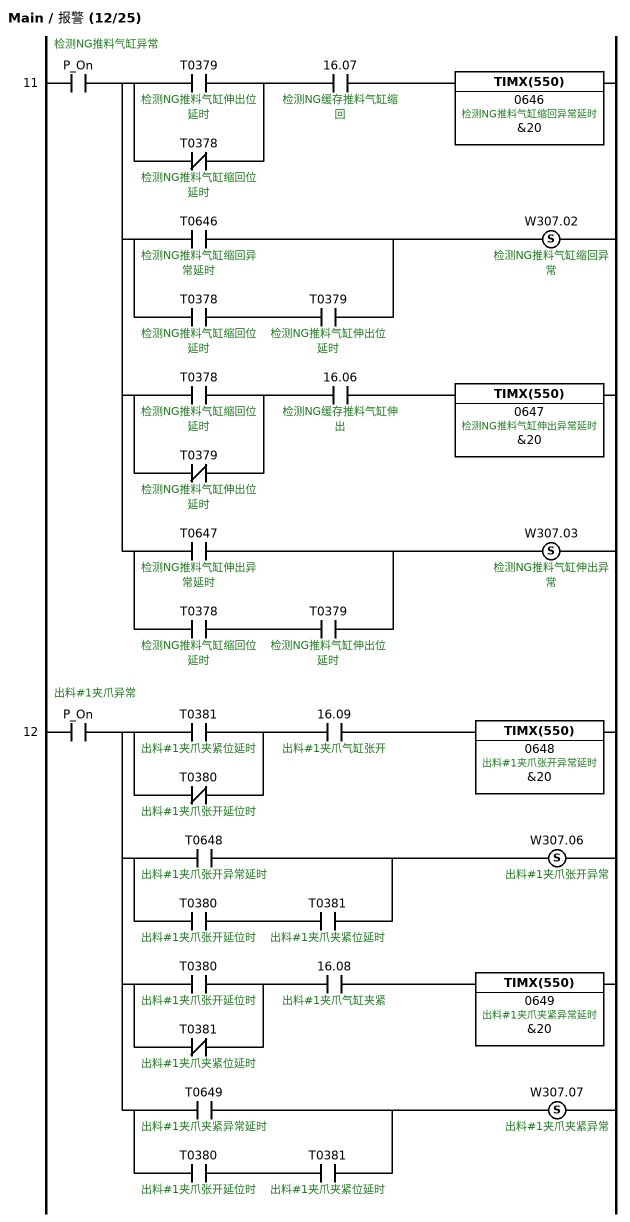
; [picture p48: Main / 报警, rungs 11-12]
; rung 11: 检测NG推料气缸异常
LD P_On
OUT TR0
LD T0379  ; 检测NG推料气缸伸出位延时
ORNOT T0378  ; 检测NG推料气缸缩回位延时
ANDLD
AND 16.07  ; 检测NG缓存推料气缸缩回
TIMX(550) 0646 &20  ; 检测NG推料气缸缩回异常延时
LD TR0
LD T0646  ; 检测NG推料气缸缩回异常延时
LD T0378  ; 检测NG推料气缸缩回位延时
AND T0379  ; 检测NG推料气缸伸出位延时
ORLD
ANDLD
SET W307.02  ; 检测NG推料气缸缩回异常
LD TR0
LD T0378  ; 检测NG推料气缸缩回位延时
ORNOT T0379  ; 检测NG推料气缸伸出位延时
ANDLD
AND 16.06  ; 检测NG缓存推料气缸伸出
TIMX(550) 0647 &20  ; 检测NG推料气缸伸出异常延时
LD TR0
LD T0647  ; 检测NG推料气缸伸出异常延时
LD T0378  ; 检测NG推料气缸缩回位延时
AND T0379  ; 检测NG推料气缸伸出位延时
ORLD
ANDLD
SET W307.03  ; 检测NG推料气缸伸出异常
; rung 12: 出料#1夹爪异常
LD P_On
OUT TR0
LD T0381  ; 出料#1夹爪夹紧位延时
ORNOT T0380  ; 出料#1夹爪张开延位时
ANDLD
AND 16.09  ; 出料#1夹爪气缸张开
TIMX(550) 0648 &20  ; 出料#1夹爪张开异常延时
LD TR0
LD T0648  ; 出料#1夹爪张开异常延时
LD T0380  ; 出料#1夹爪张开延位时
AND T0381  ; 出料#1夹爪夹紧位延时
ORLD
ANDLD
SET W307.06  ; 出料#1夹爪张开异常
LD TR0
LD T0380  ; 出料#1夹爪张开延位时
ORNOT T0381  ; 出料#1夹爪夹紧位延时
ANDLD
AND 16.08  ; 出料#1夹爪气缸夹紧
TIMX(550) 0649 &20  ; 出料#1夹爪夹紧异常延时
LD TR0
LD T0649  ; 出料#1夹爪夹紧异常延时
LD T0380  ; 出料#1夹爪张开延位时
AND T0381  ; 出料#1夹爪夹紧位延时
ORLD
ANDLD
SET W307.07  ; 出料#1夹爪夹紧异常

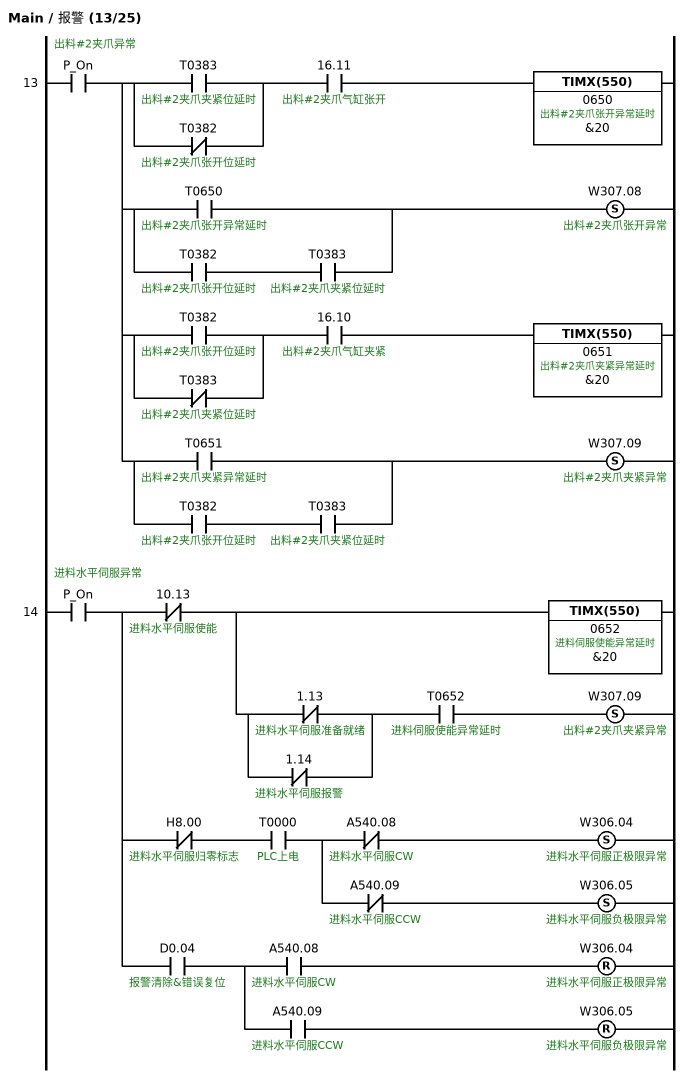
; rung 13: 出料#2夹爪异常
LD P_On
OUT TR0
LD T0383  ; 出料#2夹爪夹紧位延时
ORNOT T0382  ; 出料#2夹爪张开位延时
ANDLD
AND 16.11  ; 出料#2夹爪气缸张开
TIMX(550) 0650 &20  ; 出料#2夹爪张开异常延时
LD TR0
LD T0650  ; 出料#2夹爪张开异常延时
LD T0382  ; 出料#2夹爪张开位延时
AND T0383  ; 出料#2夹爪夹紧位延时
ORLD
ANDLD
SET W307.08  ; 出料#2夹爪张开异常
LD TR0
LD T0382  ; 出料#2夹爪张开位延时
ORNOT T0383  ; 出料#2夹爪夹紧位延时
ANDLD
AND 16.10  ; 出料#2夹爪气缸夹紧
TIMX(550) 0651 &20  ; 出料#2夹爪夹紧异常延时
LD TR0
LD T0651  ; 出料#2夹爪夹紧异常延时
LD T0382  ; 出料#2夹爪张开位延时
AND T0383  ; 出料#2夹爪夹紧位延时
ORLD
ANDLD
SET W307.09  ; 出料#2夹爪夹紧异常
; rung 14: 进料水平伺服异常
LD P_On
OUT TR0
ANDNOT 10.13  ; 进料水平伺服使能
TIMX(550) 0652 &20  ; 进料伺服使能异常延时
LDNOT 1.13  ; 进料水平伺服准备就绪
ORNOT 1.14  ; 进料水平伺服报警
ANDLD
AND T0652  ; 进料伺服使能异常延时
SET W307.09  ; 出料#2夹爪夹紧异常
LD TR0
ANDNOT H8.00  ; 进料水平伺服归零标志
AND T0000  ; PLC上电
OUT TR1
ANDNOT A540.08  ; 进料水平伺服CW
SET W306.04  ; 进料水平伺服正极限异常
LD TR1
ANDNOT A540.09  ; 进料水平伺服CCW
SET W306.05  ; 进料水平伺服负极限异常
LD TR0
AND D0.04  ; 报警清除&错误复位
OUT TR0
AND A540.08  ; 进料水平伺服CW
RSET W306.04  ; 进料水平伺服正极限异常
LD TR0
AND A540.09  ; 进料水平伺服CCW
RSET W306.05  ; 进料水平伺服负极限异常

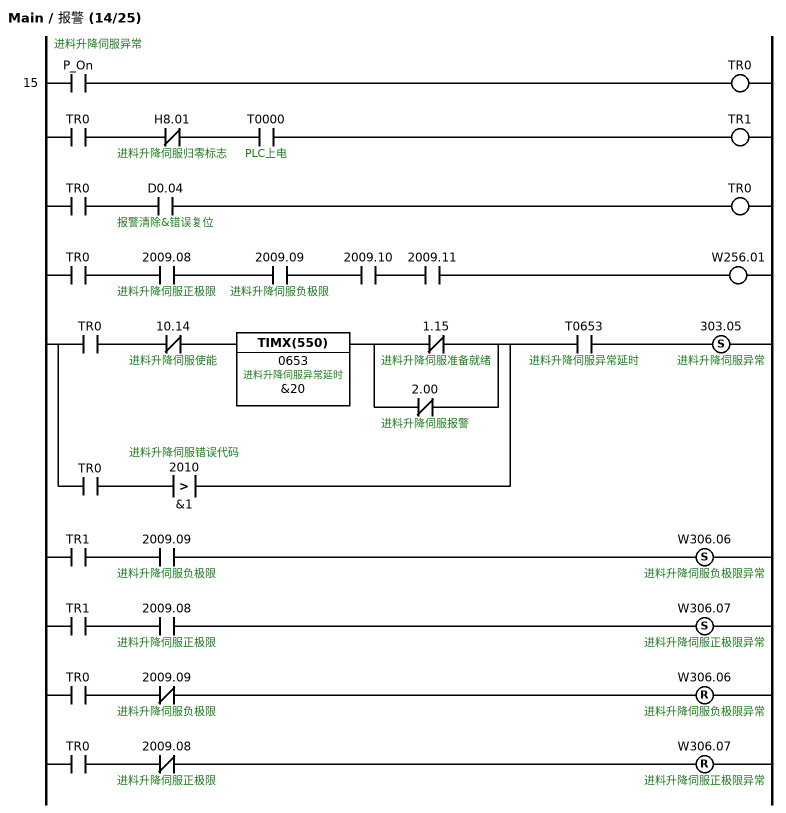
; rung 15: 进料升降伺服异常
LD P_On
OUT TR0
AND 2009.08  ; 进料升降伺服正极限
AND 2009.09  ; 进料升降伺服负极限
AND 2009.10
AND 2009.11
OUT W256.01
LD TR0
ANDNOT 10.14  ; 进料升降伺服使能
TIMX(550) 0653 &20  ; 进料升降伺服异常延时
LDNOT 1.15  ; 进料升降伺服准备就绪
ORNOT 2.00  ; 进料升降伺服报警
ANDLD
LD TR0
AND>(320) 2010 &1  ; 进料升降伺服错误代码
ORLD
AND T0653  ; 进料升降伺服异常延时
SET 303.05  ; 进料升降伺服异常
LD TR0
ANDNOT H8.01  ; 进料升降伺服归零标志
AND T0000  ; PLC上电
OUT TR1
AND 2009.09  ; 进料升降伺服负极限
SET W306.06  ; 进料升降伺服负极限异常
LD TR1
AND 2009.08  ; 进料升降伺服正极限
SET W306.07  ; 进料升降伺服正极限异常
LD TR0
AND D0.04  ; 报警清除&错误复位
OUT TR0
ANDNOT 2009.09  ; 进料升降伺服负极限
RSET W306.06  ; 进料升降伺服负极限异常
LD TR0
ANDNOT 2009.08  ; 进料升降伺服正极限
RSET W306.07  ; 进料升降伺服正极限异常

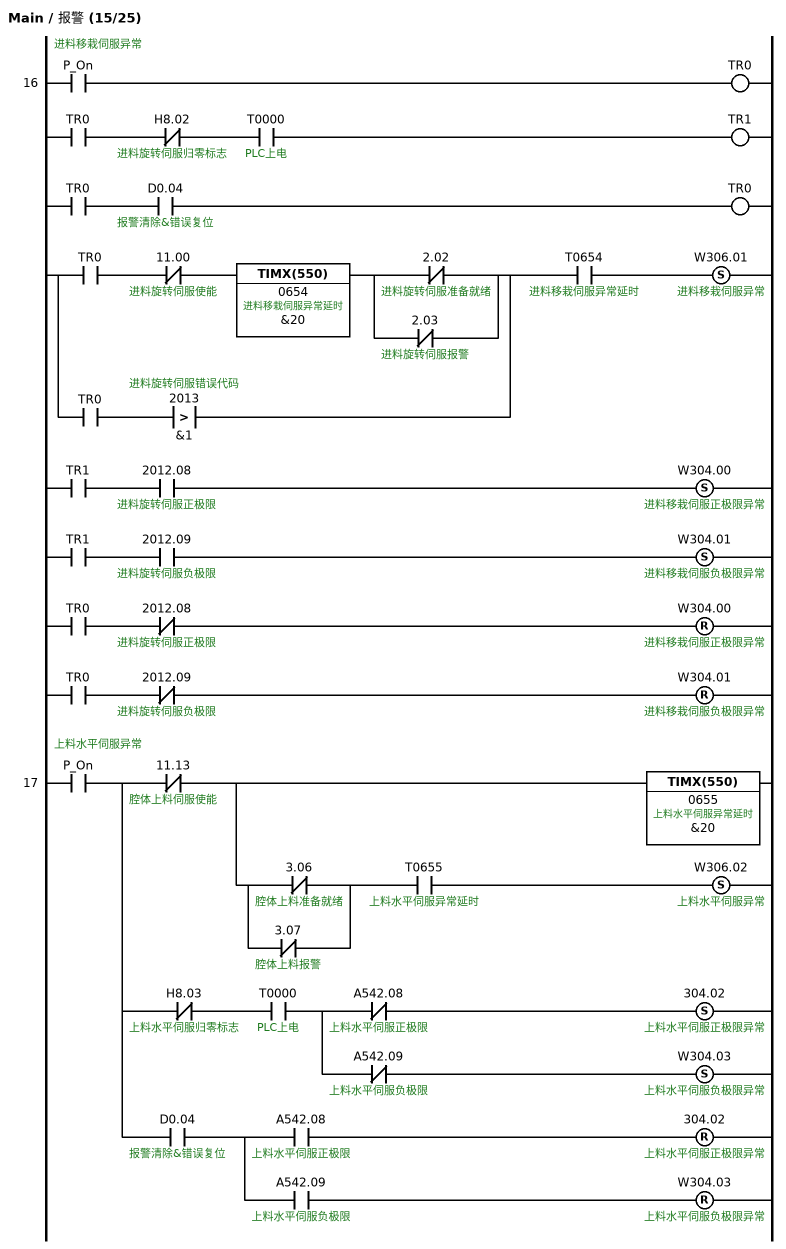
; rung 16: 进料移栽伺服异常
LD P_On
OUT TR0
ANDNOT 11.00  ; 进料旋转伺服使能
TIMX(550) 0654 &20  ; 进料移栽伺服异常延时
LDNOT 2.02  ; 进料旋转伺服准备就绪
ORNOT 2.03  ; 进料旋转伺服报警
ANDLD
LD TR0
AND>(320) 2013 &1  ; 进料旋转伺服错误代码
ORLD
AND T0654  ; 进料移栽伺服异常延时
SET W306.01  ; 进料移栽伺服异常
LD TR0
ANDNOT H8.02  ; 进料旋转伺服归零标志
AND T0000  ; PLC上电
OUT TR1
AND 2012.08  ; 进料旋转伺服正极限
SET W304.00  ; 进料移栽伺服正极限异常
LD TR1
AND 2012.09  ; 进料旋转伺服负极限
SET W304.01  ; 进料移栽伺服负极限异常
LD TR0
AND D0.04  ; 报警清除&错误复位
OUT TR0
ANDNOT 2012.08  ; 进料旋转伺服正极限
RSET W304.00  ; 进料移栽伺服正极限异常
LD TR0
ANDNOT 2012.09  ; 进料旋转伺服负极限
RSET W304.01  ; 进料移栽伺服负极限异常
; rung 17: 上料水平伺服异常
LD P_On
OUT TR0
ANDNOT 11.13  ; 腔体上料伺服使能
TIMX(550) 0655 &20  ; 上料水平伺服异常延时
LDNOT 3.06  ; 腔体上料准备就绪
ORNOT 3.07  ; 腔体上料报警
ANDLD
AND T0655  ; 上料水平伺服异常延时
SET W306.02  ; 上料水平伺服异常
LD TR0
ANDNOT H8.03  ; 上料水平伺服归零标志
AND T0000  ; PLC上电
OUT TR1
ANDNOT A542.08  ; 上料水平伺服正极限
SET 304.02  ; 上料水平伺服正极限异常
LD TR1
ANDNOT A542.09  ; 上料水平伺服负极限
SET W304.03  ; 上料水平伺服负极限异常
LD TR0
AND D0.04  ; 报警清除&错误复位
OUT TR0
AND A542.08  ; 上料水平伺服正极限
RSET 304.02  ; 上料水平伺服正极限异常
LD TR0
AND A542.09  ; 上料水平伺服负极限
RSET W304.03  ; 上料水平伺服负极限异常

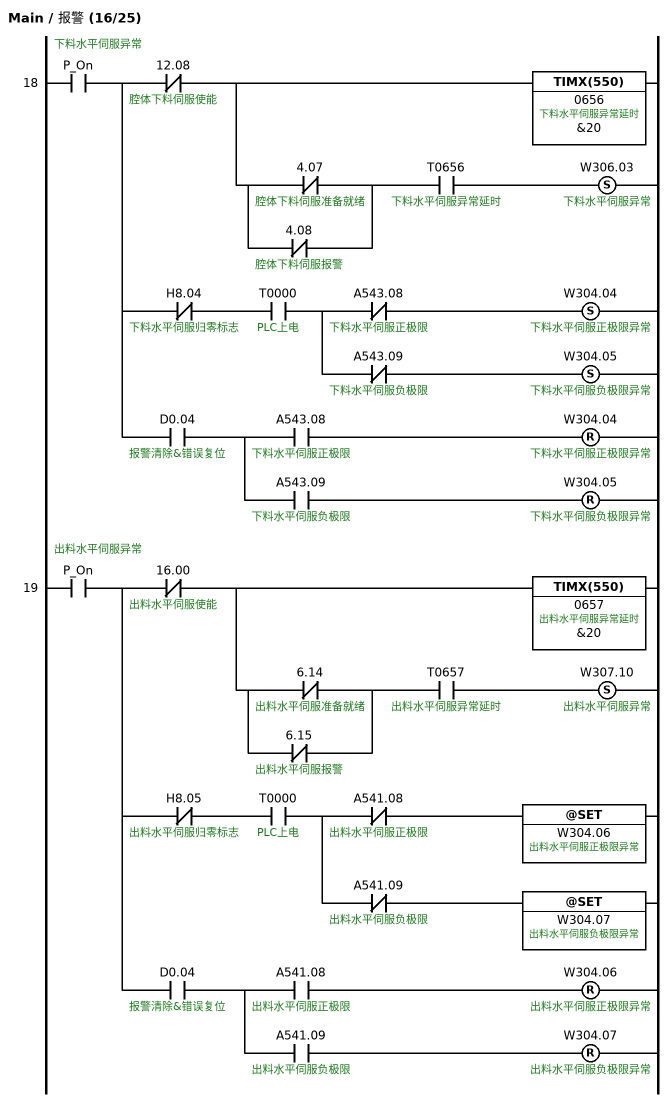
; rung 18: 下料水平伺服异常
LD P_On
OUT TR0
ANDNOT 12.08  ; 腔体下料伺服使能
TIMX(550) 0656 &20  ; 下料水平伺服异常延时
LDNOT 4.07  ; 腔体下料伺服准备就绪
ORNOT 4.08  ; 腔体下料伺服报警
ANDLD
AND T0656  ; 下料水平伺服异常延时
SET W306.03  ; 下料水平伺服异常
LD TR0
ANDNOT H8.04  ; 下料水平伺服归零标志
AND T0000  ; PLC上电
OUT TR1
ANDNOT A543.08  ; 下料水平伺服正极限
SET W304.04  ; 下料水平伺服正极限异常
LD TR1
ANDNOT A543.09  ; 下料水平伺服负极限
SET W304.05  ; 下料水平伺服负极限异常
LD TR0
AND D0.04  ; 报警清除&错误复位
OUT TR0
AND A543.08  ; 下料水平伺服正极限
RSET W304.04  ; 下料水平伺服正极限异常
LD TR0
AND A543.09  ; 下料水平伺服负极限
RSET W304.05  ; 下料水平伺服负极限异常
; rung 19: 出料水平伺服异常
LD P_On
OUT TR0
ANDNOT 16.00  ; 出料水平伺服使能
TIMX(550) 0657 &20  ; 出料水平伺服异常延时
LDNOT 6.14  ; 出料水平伺服准备就绪
ORNOT 6.15  ; 出料水平伺服报警
ANDLD
AND T0657  ; 出料水平伺服异常延时
SET W307.10  ; 出料水平伺服异常
LD TR0
ANDNOT H8.05  ; 出料水平伺服归零标志
AND T0000  ; PLC上电
OUT TR1
ANDNOT A541.08  ; 出料水平伺服正极限
@SET W304.06  ; 出料水平伺服正极限异常
LD TR1
ANDNOT A541.09  ; 出料水平伺服负极限
@SET W304.07  ; 出料水平伺服负极限异常
LD TR0
AND D0.04  ; 报警清除&错误复位
OUT TR0
AND A541.08  ; 出料水平伺服正极限
RSET W304.06  ; 出料水平伺服正极限异常
LD TR0
AND A541.09  ; 出料水平伺服负极限
RSET W304.07  ; 出料水平伺服负极限异常

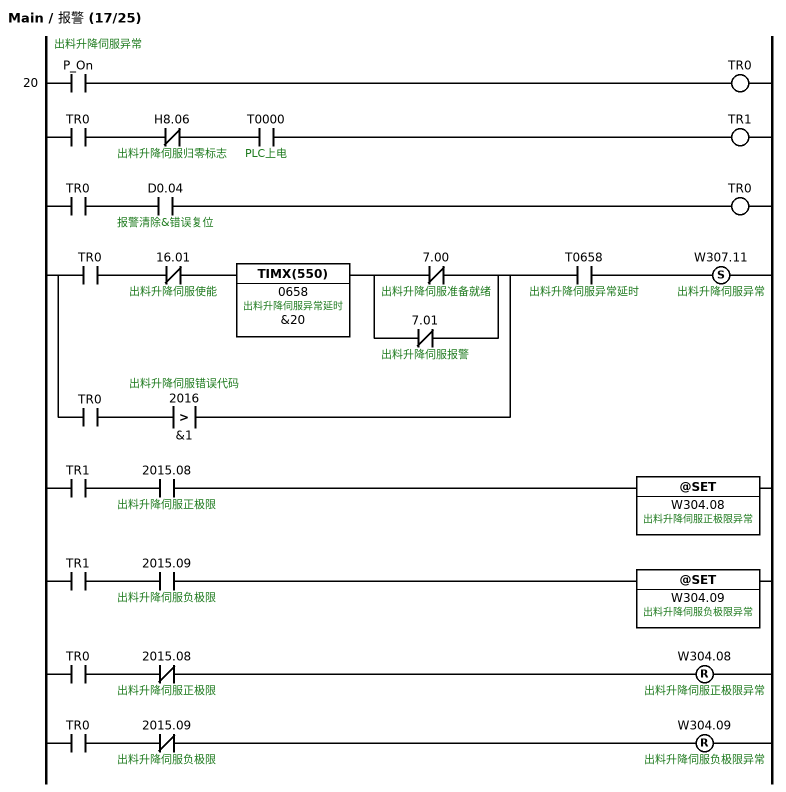
; rung 20: 出料升降伺服异常
LD P_On
OUT TR0
ANDNOT 16.01  ; 出料升降伺服使能
TIMX(550) 0658 &20  ; 出料升降伺服异常延时
LDNOT 7.00  ; 出料升降伺服准备就绪
ORNOT 7.01  ; 出料升降伺服报警
ANDLD
LD TR0
AND>(320) 2016 &1  ; 出料升降伺服错误代码
ORLD
AND T0658  ; 出料升降伺服异常延时
SET W307.11  ; 出料升降伺服异常
LD TR0
ANDNOT H8.06  ; 出料升降伺服归零标志
AND T0000  ; PLC上电
OUT TR1
AND 2015.08  ; 出料升降伺服正极限
@SET W304.08  ; 出料升降伺服正极限异常
LD TR1
AND 2015.09  ; 出料升降伺服负极限
@SET W304.09  ; 出料升降伺服负极限异常
LD TR0
AND D0.04  ; 报警清除&错误复位
OUT TR0
ANDNOT 2015.08  ; 出料升降伺服正极限
RSET W304.08  ; 出料升降伺服正极限异常
LD TR0
ANDNOT 2015.09  ; 出料升降伺服负极限
RSET W304.09  ; 出料升降伺服负极限异常

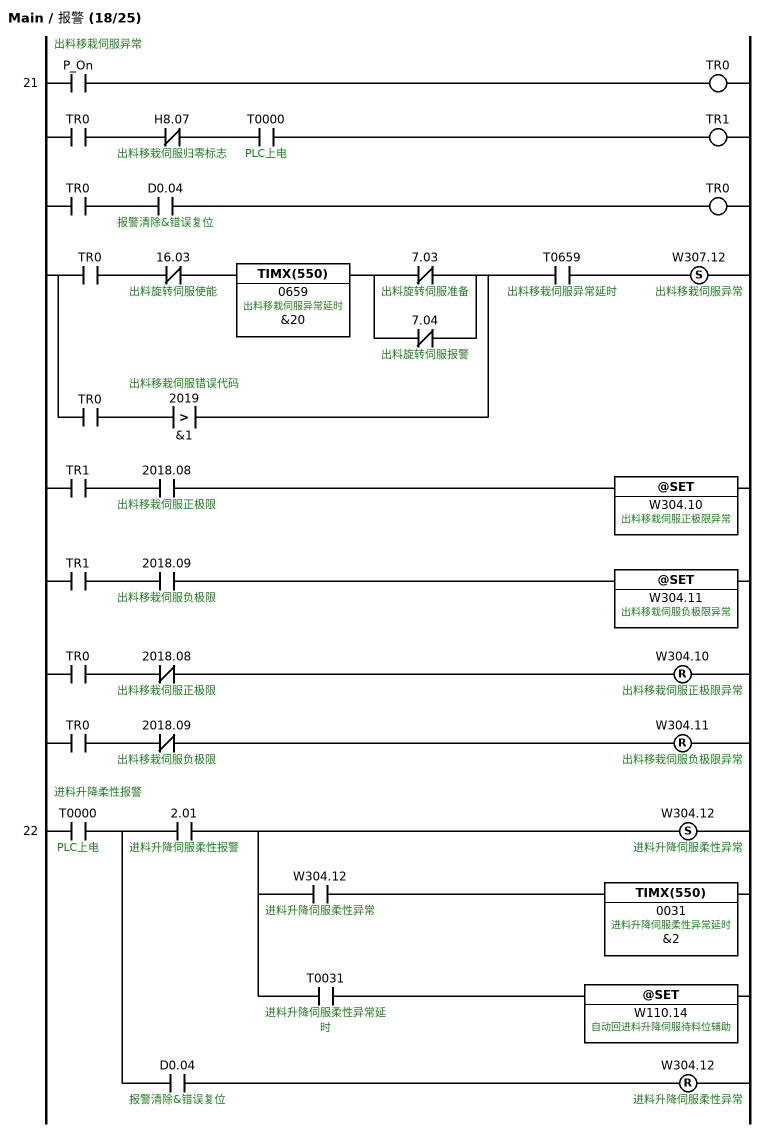
; rung 21: 出料移栽伺服异常
LD P_On
OUT TR0
ANDNOT 16.03  ; 出料旋转伺服使能
TIMX(550) 0659 &20  ; 出料移栽伺服异常延时
LDNOT 7.03  ; 出料旋转伺服准备
ORNOT 7.04  ; 出料旋转伺服报警
ANDLD
LD TR0
AND>(320) 2019 &1  ; 出料移栽伺服错误代码
ORLD
AND T0659  ; 出料移栽伺服异常延时
SET W307.12  ; 出料移栽伺服异常
LD TR0
ANDNOT H8.07  ; 出料移栽伺服归零标志
AND T0000  ; PLC上电
OUT TR1
AND 2018.08  ; 出料移栽伺服正极限
@SET W304.10  ; 出料移栽伺服正极限异常
LD TR1
AND 2018.09  ; 出料移栽伺服负极限
@SET W304.11  ; 出料移栽伺服负极限异常
LD TR0
AND D0.04  ; 报警清除&错误复位
OUT TR0
ANDNOT 2018.08  ; 出料移栽伺服正极限
RSET W304.10  ; 出料移栽伺服正极限异常
LD TR0
ANDNOT 2018.09  ; 出料移栽伺服负极限
RSET W304.11  ; 出料移栽伺服负极限异常
; rung 22: 进料升降柔性报警
LD T0000  ; PLC上电
OUT TR0
AND 2.01  ; 进料升降伺服柔性报警
OUT TR1
SET W304.12  ; 进料升降伺服柔性异常
AND W304.12  ; 进料升降伺服柔性异常
TIMX(550) 0031 &2  ; 进料升降伺服柔性异常延时
LD TR1
AND T0031  ; 进料升降伺服柔性异常延时
@SET W110.14  ; 自动回进料升降伺服待料位辅助
LD TR0
AND D0.04  ; 报警清除&错误复位
RSET W304.12  ; 进料升降伺服柔性异常

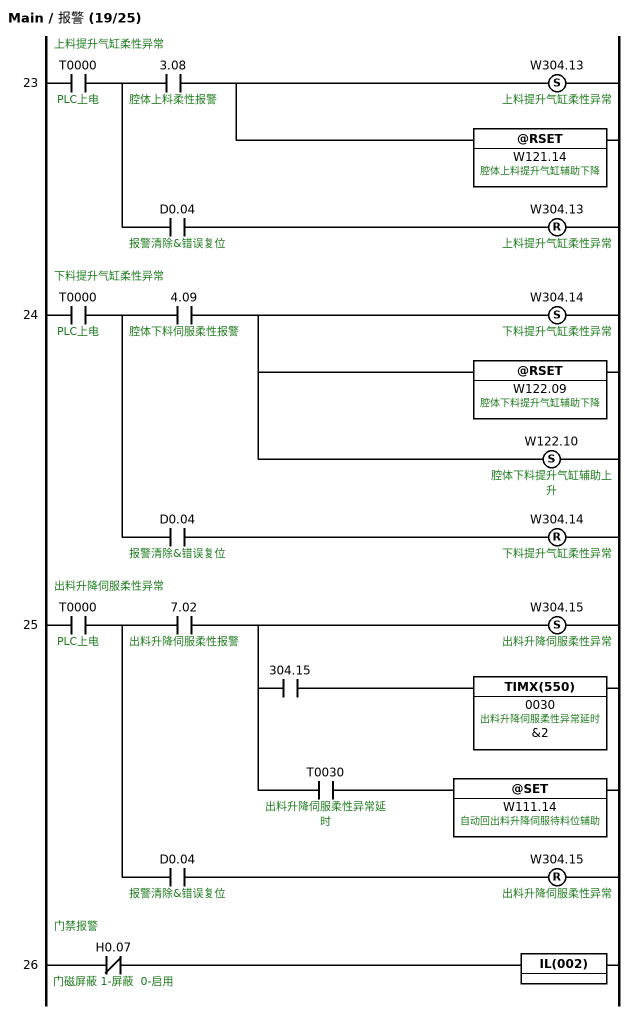
; rung 23: 上料提升气缸柔性异常
LD T0000  ; PLC上电
OUT TR0
AND 3.08  ; 腔体上料柔性报警
SET W304.13  ; 上料提升气缸柔性异常
@RSET W121.14  ; 腔体上料提升气缸辅助下降
LD TR0
AND D0.04  ; 报警清除&错误复位
RSET W304.13  ; 上料提升气缸柔性异常
; rung 24: 下料提升气缸柔性异常
LD T0000  ; PLC上电
OUT TR0
AND 4.09  ; 腔体下料伺服柔性报警
SET W304.14  ; 下料提升气缸柔性异常
@RSET W122.09  ; 腔体下料提升气缸辅助下降
SET W122.10  ; 腔体下料提升气缸辅助上升
LD TR0
AND D0.04  ; 报警清除&错误复位
RSET W304.14  ; 下料提升气缸柔性异常
; rung 25: 出料升降伺服柔性异常
LD T0000  ; PLC上电
OUT TR0
AND 7.02  ; 出料升降伺服柔性报警
OUT TR1
SET W304.15  ; 出料升降伺服柔性异常
AND 304.15
TIMX(550) 0030 &2  ; 出料升降伺服柔性异常延时
LD TR1
AND T0030  ; 出料升降伺服柔性异常延时
@SET W111.14  ; 自动回出料升降伺服待料位辅助
LD TR0
AND D0.04  ; 报警清除&错误复位
RSET W304.15  ; 出料升降伺服柔性异常
; rung 26: 门禁报警
LDNOT H0.07  ; 门磁屏蔽 1-屏蔽  0-启用
IL(002)

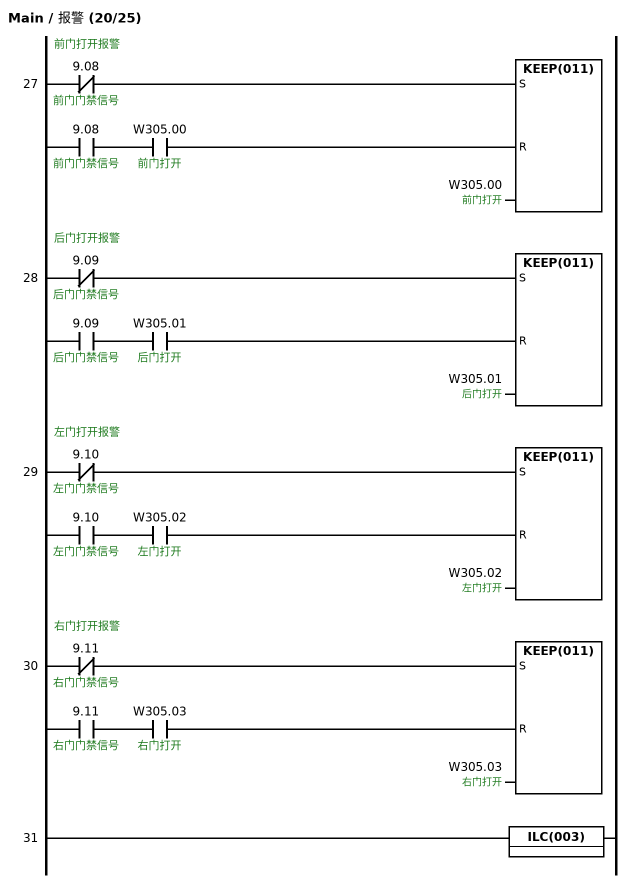
; rung 27: 前门打开报警
LDNOT 9.08  ; 前门门禁信号
LD 9.08  ; 前门门禁信号
AND W305.00  ; 前门打开
KEEP(011) W305.00  ; 前门打开
; rung 28: 后门打开报警
LDNOT 9.09  ; 后门门禁信号
LD 9.09  ; 后门门禁信号
AND W305.01  ; 后门打开
KEEP(011) W305.01  ; 后门打开
; rung 29: 左门打开报警
LDNOT 9.10  ; 左门门禁信号
LD 9.10  ; 左门门禁信号
AND W305.02  ; 左门打开
KEEP(011) W305.02  ; 左门打开
; rung 30: 右门打开报警
LDNOT 9.11  ; 右门门禁信号
LD 9.11  ; 右门门禁信号
AND W305.03  ; 右门打开
KEEP(011) W305.03  ; 右门打开
; rung 31
ILC(003)

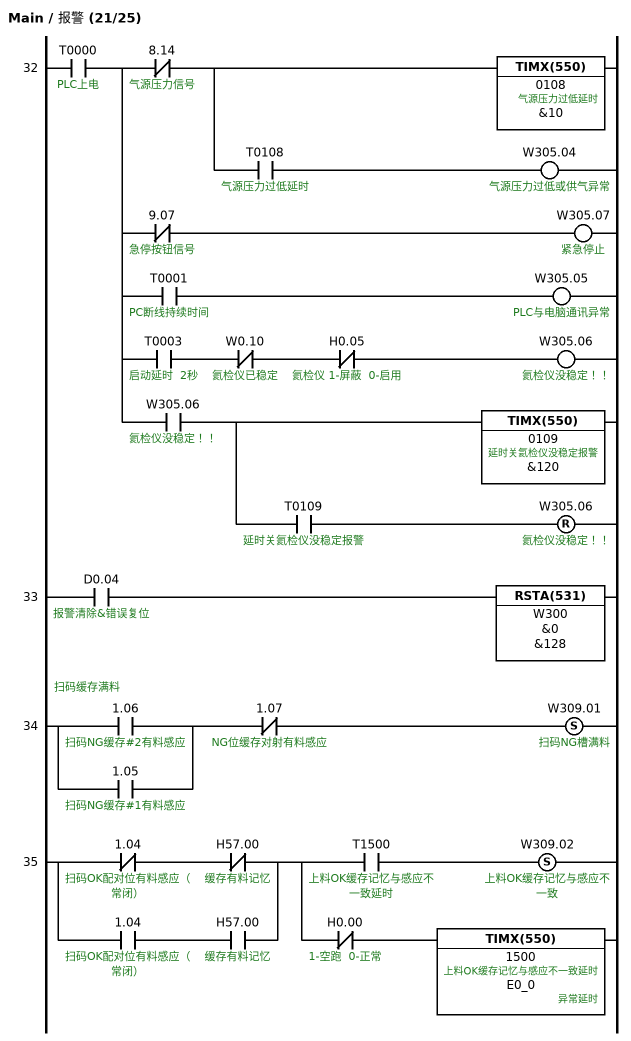
; rung 32
LD T0000  ; PLC上电
OUT TR0
ANDNOT 8.14  ; 气源压力信号
TIMX(550) 0108 &10  ; 气源压力过低延时
AND T0108  ; 气源压力过低延时
OUT W305.04  ; 气源压力过低或供气异常
LD TR0
ANDNOT 9.07  ; 急停按钮信号
OUT W305.07  ; 紧急停止
LD TR0
AND T0001  ; PC断线持续时间
OUT W305.05  ; PLC与电脑通讯异常
LD TR0
AND T0003  ; 启动延时  2秒
ANDNOT W0.10  ; 氦检仪已稳定
ANDNOT H0.05  ; 氦检仪 1-屏蔽  0-启用
OUT W305.06  ; 氦检仪没稳定！！
LD TR0
AND W305.06  ; 氦检仪没稳定！！
TIMX(550) 0109 &120  ; 延时关氦检仪没稳定报警
AND T0109  ; 延时关氦检仪没稳定报警
RSET W305.06  ; 氦检仪没稳定！！
; rung 33
LD D0.04  ; 报警清除&错误复位
RSTA(531) W300 &0 &128
; rung 34: 扫码缓存满料
LD 1.06  ; 扫码NG缓存#2有料感应
OR 1.05  ; 扫码NG缓存#1有料感应
ANDNOT 1.07  ; NG位缓存对射有料感应
SET W309.01  ; 扫码NG槽满料
; rung 35
LDNOT 1.04  ; 扫码OK配对位有料感应（常闭）
ANDNOT H57.00  ; 缓存有料记忆
LD 1.04  ; 扫码OK配对位有料感应（常闭）
AND H57.00  ; 缓存有料记忆
ORLD
OUT TR0
AND T1500  ; 上料OK缓存记忆与感应不一致延时
SET W309.02  ; 上料OK缓存记忆与感应不一致
LD TR0
ANDNOT H0.00  ; 1-空跑  0-正常
TIMX(550) 1500 E0_0  ; 异常延时, 上料OK缓存记忆与感应不一致延时

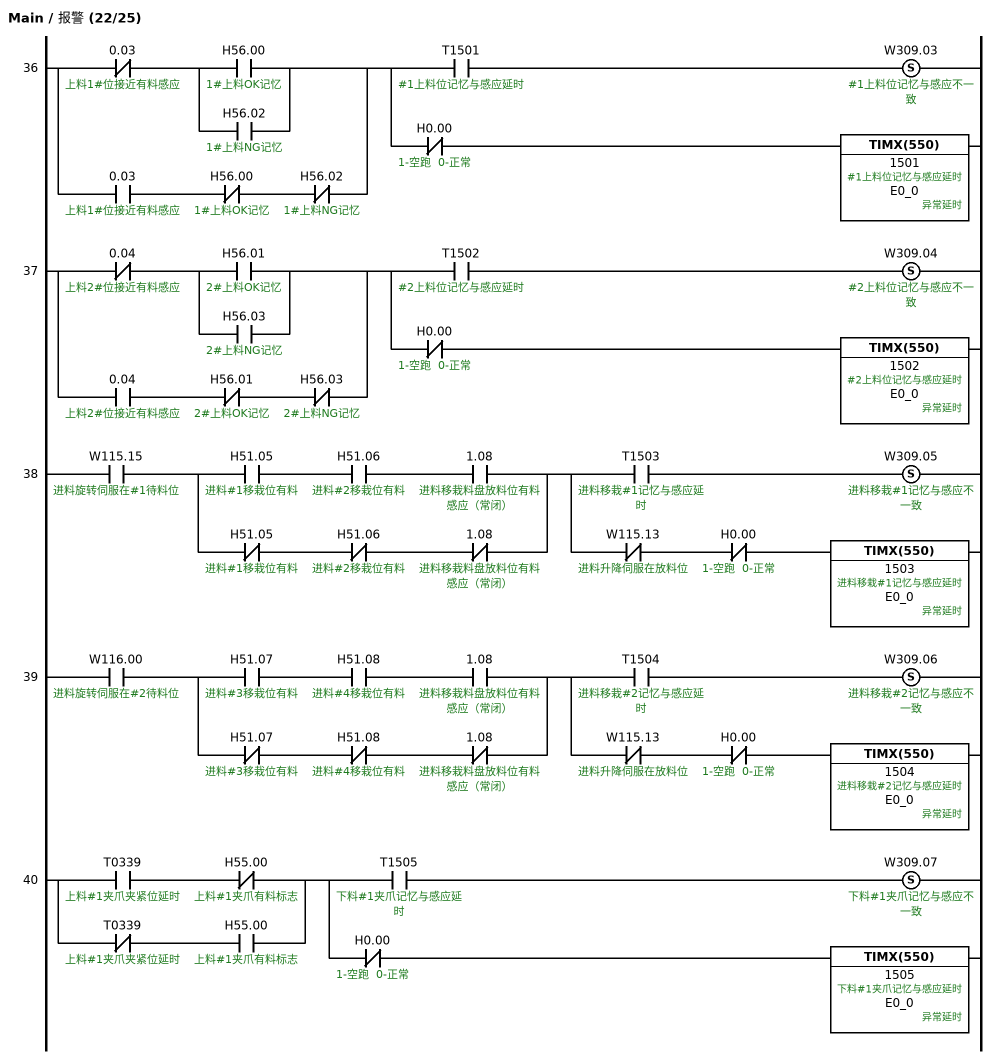
; rung 36
LDNOT 0.03  ; 上料1#位接近有料感应
LD H56.00  ; 1#上料OK记忆
OR H56.02  ; 1#上料NG记忆
ANDLD
LD 0.03  ; 上料1#位接近有料感应
ANDNOT H56.00  ; 1#上料OK记忆
ANDNOT H56.02  ; 1#上料NG记忆
ORLD
OUT TR0
AND T1501  ; #1上料位记忆与感应延时
SET W309.03  ; #1上料位记忆与感应不一致
LD TR0
ANDNOT H0.00  ; 1-空跑  0-正常
TIMX(550) 1501 E0_0  ; 异常延时, #1上料位记忆与感应延时
; rung 37
LDNOT 0.04  ; 上料2#位接近有料感应
LD H56.01  ; 2#上料OK记忆
OR H56.03  ; 2#上料NG记忆
ANDLD
LD 0.04  ; 上料2#位接近有料感应
ANDNOT H56.01  ; 2#上料OK记忆
ANDNOT H56.03  ; 2#上料NG记忆
ORLD
OUT TR0
AND T1502  ; #2上料位记忆与感应延时
SET W309.04  ; #2上料位记忆与感应不一致
LD TR0
ANDNOT H0.00  ; 1-空跑  0-正常
TIMX(550) 1502 E0_0  ; 异常延时, #2上料位记忆与感应延时
; rung 38
LD W115.15  ; 进料旋转伺服在#1待料位
LD H51.05  ; 进料#1移栽位有料
AND H51.06  ; 进料#2移栽位有料
AND 1.08  ; 进料移栽料盘放料位有料感应（常闭）
LDNOT H51.05  ; 进料#1移栽位有料
ANDNOT H51.06  ; 进料#2移栽位有料
ANDNOT 1.08  ; 进料移栽料盘放料位有料感应（常闭）
ORLD
ANDLD
OUT TR0
AND T1503  ; 进料移栽#1记忆与感应延时
SET W309.05  ; 进料移栽#1记忆与感应不一致
LD TR0
ANDNOT W115.13  ; 进料升降伺服在放料位
ANDNOT H0.00  ; 1-空跑  0-正常
TIMX(550) 1503 E0_0  ; 异常延时, 进料移栽#1记忆与感应延时
; rung 39
LD W116.00  ; 进料旋转伺服在#2待料位
LD H51.07  ; 进料#3移栽位有料
AND H51.08  ; 进料#4移栽位有料
AND 1.08  ; 进料移栽料盘放料位有料感应（常闭）
LDNOT H51.07  ; 进料#3移栽位有料
ANDNOT H51.08  ; 进料#4移栽位有料
ANDNOT 1.08  ; 进料移栽料盘放料位有料感应（常闭）
ORLD
ANDLD
OUT TR0
AND T1504  ; 进料移栽#2记忆与感应延时
SET W309.06  ; 进料移栽#2记忆与感应不一致
LD TR0
ANDNOT W115.13  ; 进料升降伺服在放料位
ANDNOT H0.00  ; 1-空跑  0-正常
TIMX(550) 1504 E0_0  ; 异常延时, 进料移栽#2记忆与感应延时
; rung 40
LD T0339  ; 上料#1夹爪夹紧位延时
ANDNOT H55.00  ; 上料#1夹爪有料标志
LDNOT T0339  ; 上料#1夹爪夹紧位延时
AND H55.00  ; 上料#1夹爪有料标志
ORLD
OUT TR0
AND T1505  ; 下料#1夹爪记忆与感应延时
SET W309.07  ; 下料#1夹爪记忆与感应不一致
LD TR0
ANDNOT H0.00  ; 1-空跑  0-正常
TIMX(550) 1505 E0_0  ; 异常延时, 下料#1夹爪记忆与感应延时

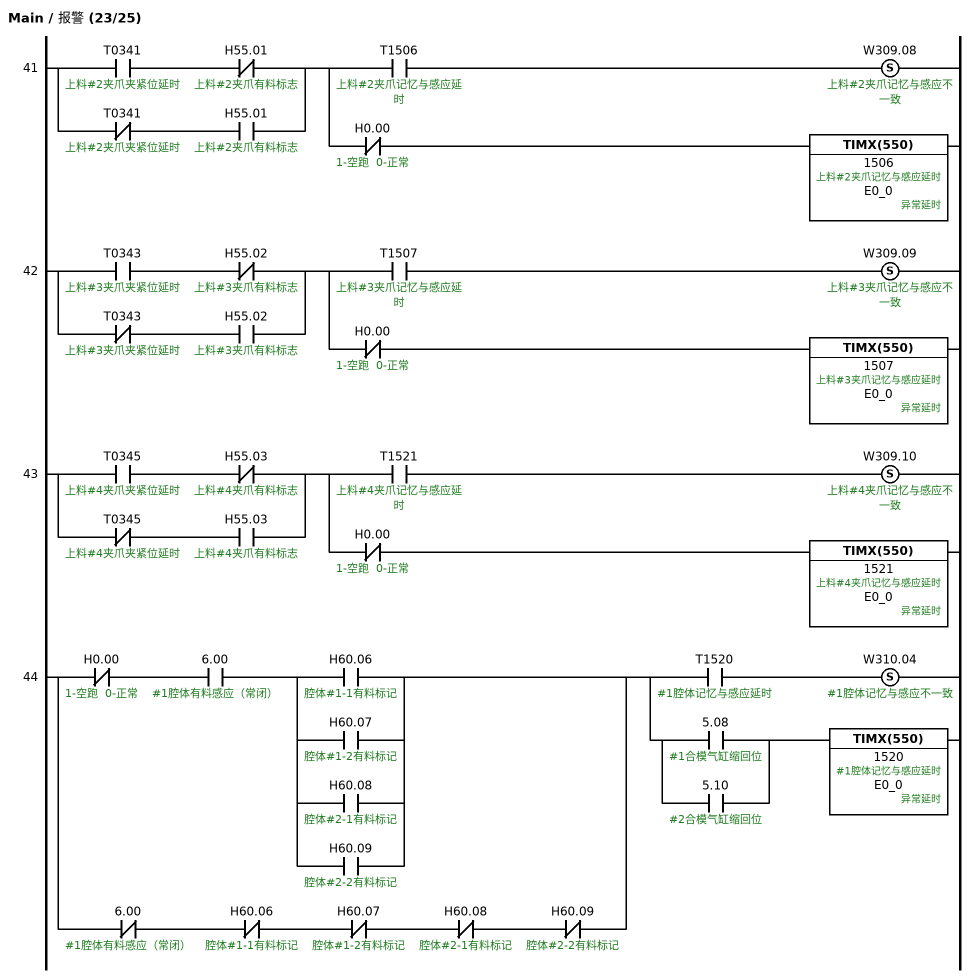
; rung 41
LD T0341  ; 上料#2夹爪夹紧位延时
ANDNOT H55.01  ; 上料#2夹爪有料标志
LDNOT T0341  ; 上料#2夹爪夹紧位延时
AND H55.01  ; 上料#2夹爪有料标志
ORLD
OUT TR0
AND T1506  ; 上料#2夹爪记忆与感应延时
SET W309.08  ; 上料#2夹爪记忆与感应不一致
LD TR0
ANDNOT H0.00  ; 1-空跑  0-正常
TIMX(550) 1506 E0_0  ; 异常延时, 上料#2夹爪记忆与感应延时
; rung 42
LD T0343  ; 上料#3夹爪夹紧位延时
ANDNOT H55.02  ; 上料#3夹爪有料标志
LDNOT T0343  ; 上料#3夹爪夹紧位延时
AND H55.02  ; 上料#3夹爪有料标志
ORLD
OUT TR0
AND T1507  ; 上料#3夹爪记忆与感应延时
SET W309.09  ; 上料#3夹爪记忆与感应不一致
LD TR0
ANDNOT H0.00  ; 1-空跑  0-正常
TIMX(550) 1507 E0_0  ; 异常延时, 上料#3夹爪记忆与感应延时
; rung 43
LD T0345  ; 上料#4夹爪夹紧位延时
ANDNOT H55.03  ; 上料#4夹爪有料标志
LDNOT T0345  ; 上料#4夹爪夹紧位延时
AND H55.03  ; 上料#4夹爪有料标志
ORLD
OUT TR0
AND T1521  ; 上料#4夹爪记忆与感应延时
SET W309.10  ; 上料#4夹爪记忆与感应不一致
LD TR0
ANDNOT H0.00  ; 1-空跑  0-正常
TIMX(550) 1521 E0_0  ; 异常延时, 上料#4夹爪记忆与感应延时
; rung 44
LDNOT H0.00  ; 1-空跑  0-正常
AND 6.00  ; #1腔体有料感应（常闭）
LD H60.06  ; 腔体#1-1有料标记
OR H60.07  ; 腔体#1-2有料标记
OR H60.08  ; 腔体#2-1有料标记
OR H60.09  ; 腔体#2-2有料标记
ANDLD
LDNOT 6.00  ; #1腔体有料感应（常闭）
ANDNOT H60.06  ; 腔体#1-1有料标记
ANDNOT H60.07  ; 腔体#1-2有料标记
ANDNOT H60.08  ; 腔体#2-1有料标记
ANDNOT H60.09  ; 腔体#2-2有料标记
ORLD
OUT TR0
AND T1520  ; #1腔体记忆与感应延时
SET W310.04  ; #1腔体记忆与感应不一致
LD TR0
LD 5.08  ; #1合模气缸缩回位
OR 5.10  ; #2合模气缸缩回位
ANDLD
TIMX(550) 1520 E0_0  ; 异常延时, #1腔体记忆与感应延时

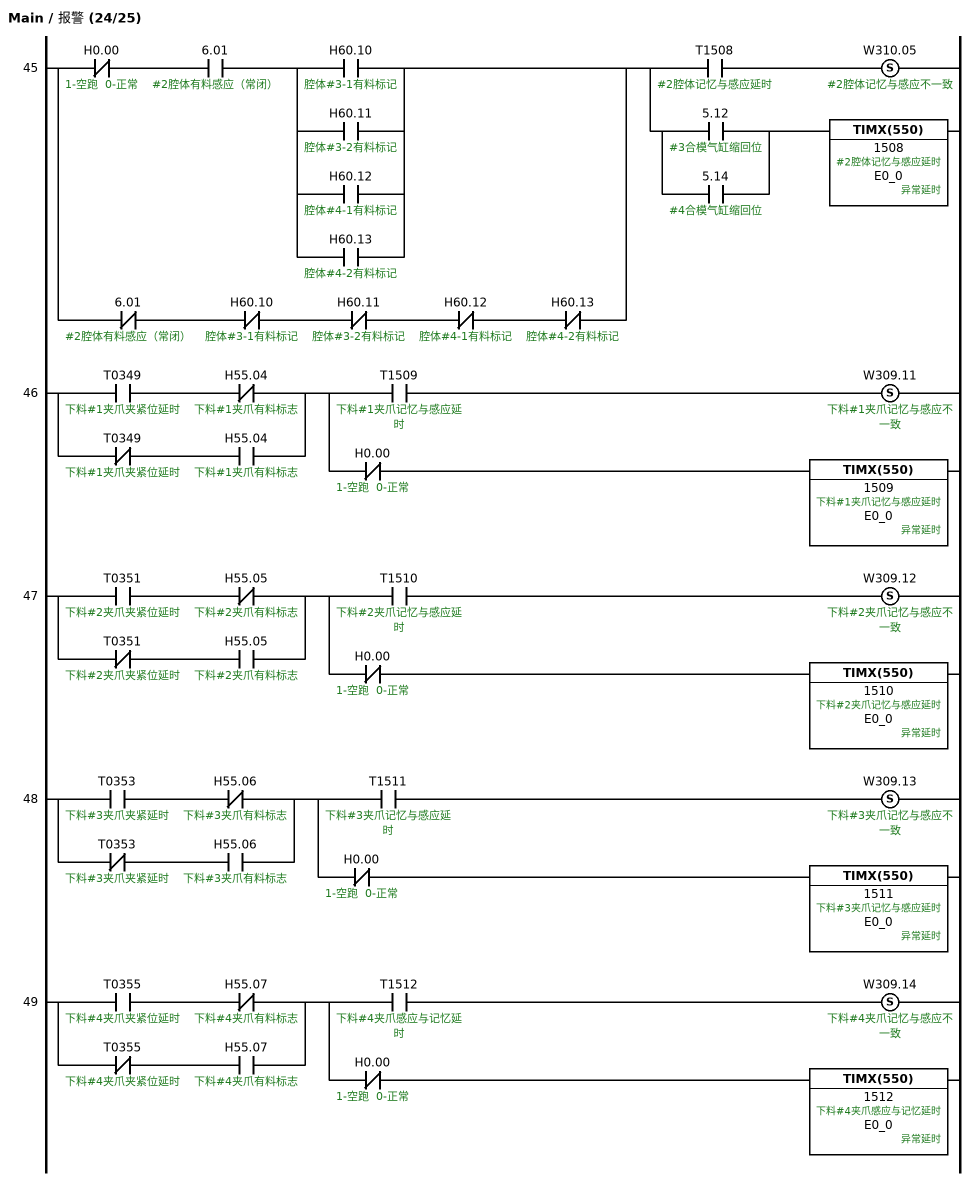
; rung 45
LDNOT H0.00  ; 1-空跑  0-正常
AND 6.01  ; #2腔体有料感应（常闭）
LD H60.10  ; 腔体#3-1有料标记
OR H60.11  ; 腔体#3-2有料标记
OR H60.12  ; 腔体#4-1有料标记
OR H60.13  ; 腔体#4-2有料标记
ANDLD
LDNOT 6.01  ; #2腔体有料感应（常闭）
ANDNOT H60.10  ; 腔体#3-1有料标记
ANDNOT H60.11  ; 腔体#3-2有料标记
ANDNOT H60.12  ; 腔体#4-1有料标记
ANDNOT H60.13  ; 腔体#4-2有料标记
ORLD
OUT TR0
AND T1508  ; #2腔体记忆与感应延时
SET W310.05  ; #2腔体记忆与感应不一致
LD TR0
LD 5.12  ; #3合模气缸缩回位
OR 5.14  ; #4合模气缸缩回位
ANDLD
TIMX(550) 1508 E0_0  ; 异常延时, #2腔体记忆与感应延时
; rung 46
LD T0349  ; 下料#1夹爪夹紧位延时
ANDNOT H55.04  ; 下料#1夹爪有料标志
LDNOT T0349  ; 下料#1夹爪夹紧位延时
AND H55.04  ; 下料#1夹爪有料标志
ORLD
OUT TR0
AND T1509  ; 下料#1夹爪记忆与感应延时
SET W309.11  ; 下料#1夹爪记忆与感应不一致
LD TR0
ANDNOT H0.00  ; 1-空跑  0-正常
TIMX(550) 1509 E0_0  ; 异常延时, 下料#1夹爪记忆与感应延时
; rung 47
LD T0351  ; 下料#2夹爪夹紧位延时
ANDNOT H55.05  ; 下料#2夹爪有料标志
LDNOT T0351  ; 下料#2夹爪夹紧位延时
AND H55.05  ; 下料#2夹爪有料标志
ORLD
OUT TR0
AND T1510  ; 下料#2夹爪记忆与感应延时
SET W309.12  ; 下料#2夹爪记忆与感应不一致
LD TR0
ANDNOT H0.00  ; 1-空跑  0-正常
TIMX(550) 1510 E0_0  ; 异常延时, 下料#2夹爪记忆与感应延时
; rung 48
LD T0353  ; 下料#3夹爪夹紧延时
ANDNOT H55.06  ; 下料#3夹爪有料标志
LDNOT T0353  ; 下料#3夹爪夹紧延时
AND H55.06  ; 下料#3夹爪有料标志
ORLD
OUT TR0
AND T1511  ; 下料#3夹爪记忆与感应延时
SET W309.13  ; 下料#3夹爪记忆与感应不一致
LD TR0
ANDNOT H0.00  ; 1-空跑  0-正常
TIMX(550) 1511 E0_0  ; 异常延时, 下料#3夹爪记忆与感应延时
; rung 49
LD T0355  ; 下料#4夹爪夹紧位延时
ANDNOT H55.07  ; 下料#4夹爪有料标志
LDNOT T0355  ; 下料#4夹爪夹紧位延时
AND H55.07  ; 下料#4夹爪有料标志
ORLD
OUT TR0
AND T1512  ; 下料#4夹爪感应与记忆延时
SET W309.14  ; 下料#4夹爪记忆与感应不一致
LD TR0
ANDNOT H0.00  ; 1-空跑  0-正常
TIMX(550) 1512 E0_0  ; 异常延时, 下料#4夹爪感应与记忆延时

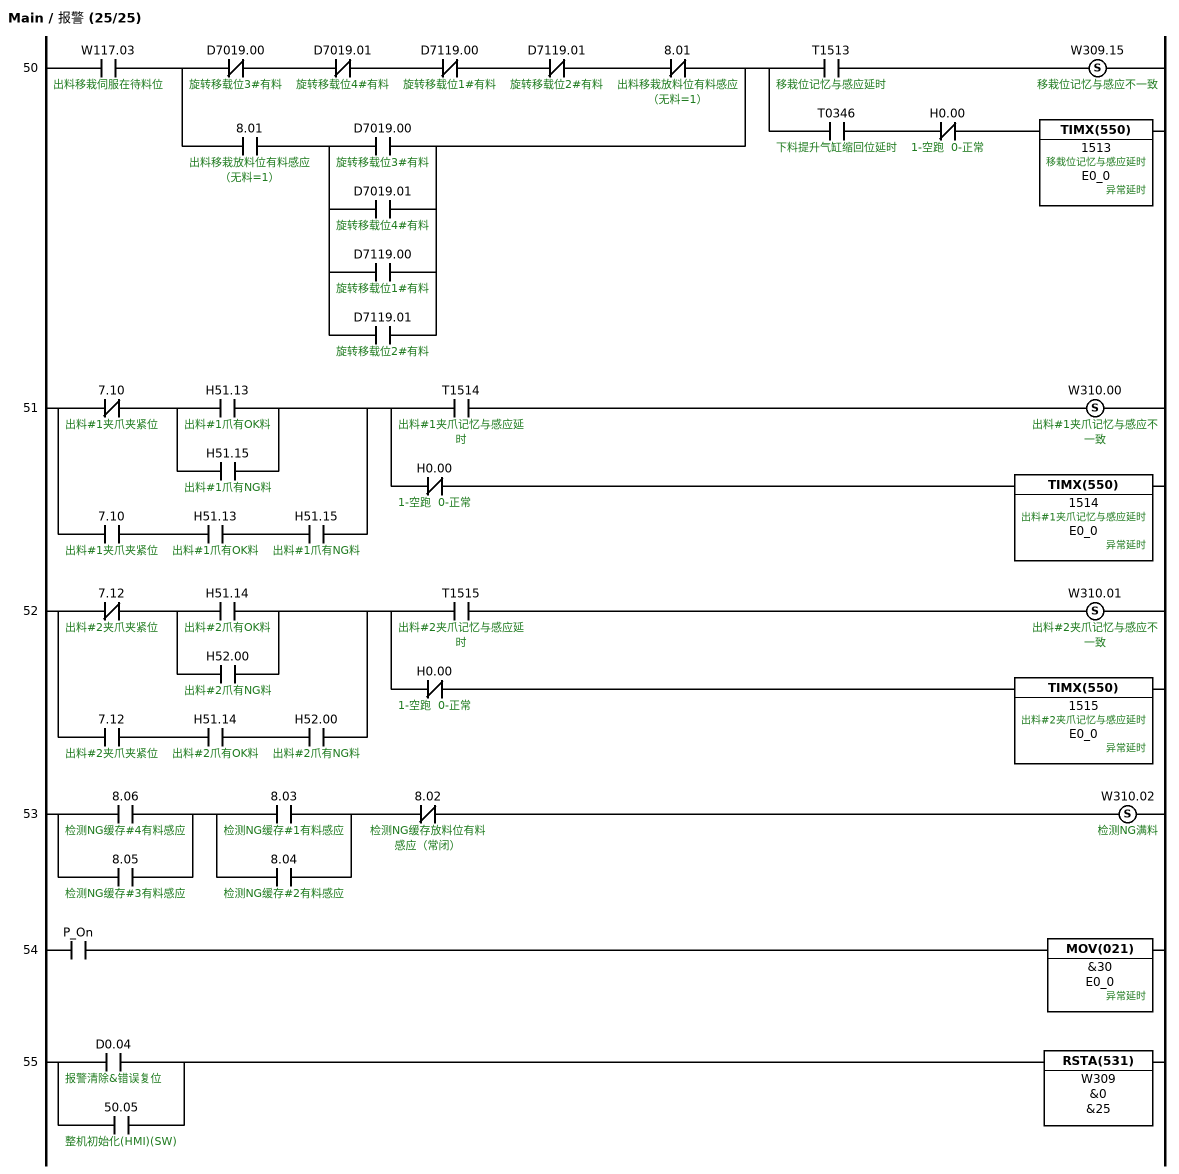
; rung 50
LD W117.03  ; 出料移栽伺服在待料位
LDNOT D7019.00  ; 旋转移载位3#有料
ANDNOT D7019.01  ; 旋转移载位4#有料
ANDNOT D7119.00  ; 旋转移载位1#有料
ANDNOT D7119.01  ; 旋转移载位2#有料
ANDNOT 8.01  ; 出料移栽放料位有料感应（无料=1）
LD 8.01  ; 出料移栽放料位有料感应（无料=1）
LD D7019.00  ; 旋转移载位3#有料
OR D7019.01  ; 旋转移载位4#有料
OR D7119.00  ; 旋转移载位1#有料
OR D7119.01  ; 旋转移载位2#有料
ANDLD
ORLD
ANDLD
OUT TR0
AND T1513  ; 移栽位记忆与感应延时
SET W309.15  ; 移栽位记忆与感应不一致
LD TR0
AND T0346  ; 下料提升气缸缩回位延时
ANDNOT H0.00  ; 1-空跑  0-正常
TIMX(550) 1513 E0_0  ; 异常延时, 移栽位记忆与感应延时
; rung 51
LDNOT 7.10  ; 出料#1夹爪夹紧位
LD H51.13  ; 出料#1爪有OK料
OR H51.15  ; 出料#1爪有NG料
ANDLD
LD 7.10  ; 出料#1夹爪夹紧位
AND H51.13  ; 出料#1爪有OK料
AND H51.15  ; 出料#1爪有NG料
ORLD
OUT TR0
AND T1514  ; 出料#1夹爪记忆与感应延时
SET W310.00  ; 出料#1夹爪记忆与感应不一致
LD TR0
ANDNOT H0.00  ; 1-空跑  0-正常
TIMX(550) 1514 E0_0  ; 异常延时, 出料#1夹爪记忆与感应延时
; rung 52
LDNOT 7.12  ; 出料#2夹爪夹紧位
LD H51.14  ; 出料#2爪有OK料
OR H52.00  ; 出料#2爪有NG料
ANDLD
LD 7.12  ; 出料#2夹爪夹紧位
AND H51.14  ; 出料#2爪有OK料
AND H52.00  ; 出料#2爪有NG料
ORLD
OUT TR0
AND T1515  ; 出料#2夹爪记忆与感应延时
SET W310.01  ; 出料#2夹爪记忆与感应不一致
LD TR0
ANDNOT H0.00  ; 1-空跑  0-正常
TIMX(550) 1515 E0_0  ; 异常延时, 出料#2夹爪记忆与感应延时
; rung 53
LD 8.06  ; 检测NG缓存#4有料感应
OR 8.05  ; 检测NG缓存#3有料感应
LD 8.03  ; 检测NG缓存#1有料感应
OR 8.04  ; 检测NG缓存#2有料感应
ANDLD
ANDNOT 8.02  ; 检测NG缓存放料位有料感应（常闭）
SET W310.02  ; 检测NG满料
; rung 54
LD P_On
MOV(021) &30 E0_0  ; 异常延时
; rung 55
LD D0.04  ; 报警清除&错误复位
OR 50.05  ; 整机初始化(HMI)(SW)
RSTA(531) W309 &0 &25

### Section 复位

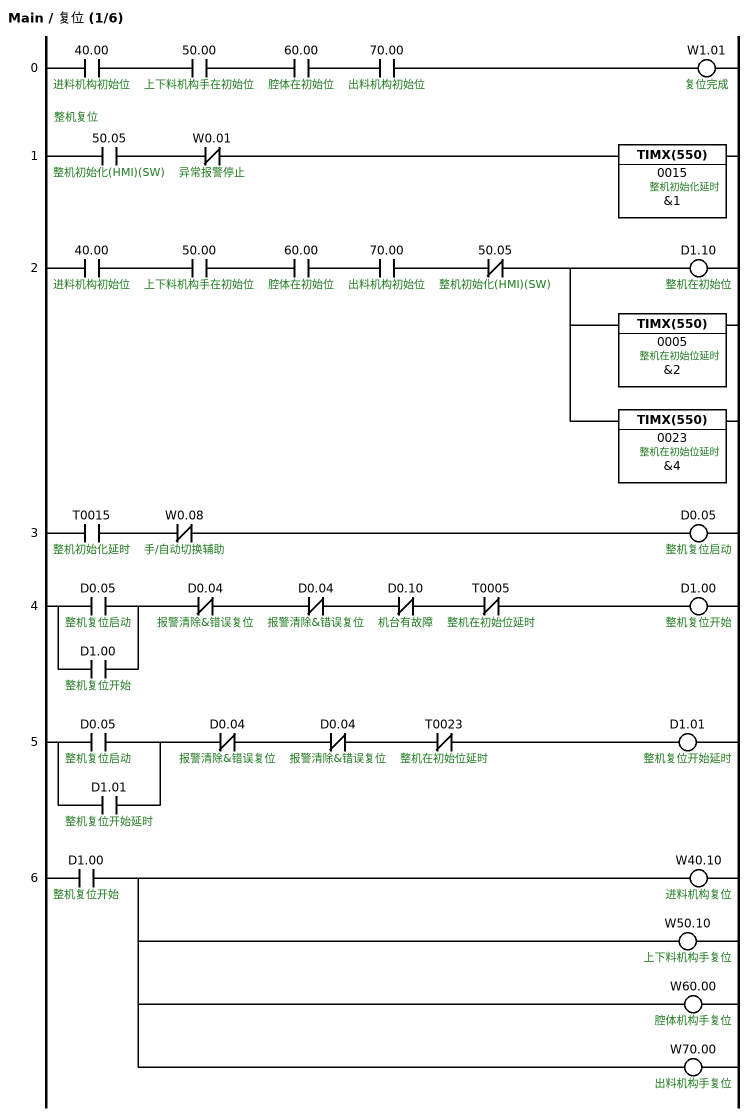
; rung 0
LD 40.00  ; 进料机构初始位
AND 50.00  ; 上下料机构手在初始位
AND 60.00  ; 腔体在初始位
AND 70.00  ; 出料机构初始位
OUT W1.01  ; 复位完成
; rung 1: 整机复位
LD 50.05  ; 整机初始化(HMI)(SW)
ANDNOT W0.01  ; 异常报警停止
TIMX(550) 0015 &1  ; 整机初始化延时
; rung 2
LD 40.00  ; 进料机构初始位
AND 50.00  ; 上下料机构手在初始位
AND 60.00  ; 腔体在初始位
AND 70.00  ; 出料机构初始位
ANDNOT 50.05  ; 整机初始化(HMI)(SW)
OUT D1.10  ; 整机在初始位
TIMX(550) 0005 &2  ; 整机在初始位延时
TIMX(550) 0023 &4  ; 整机在初始位延时
; rung 3
LD T0015  ; 整机初始化延时
ANDNOT W0.08  ; 手/自动切换辅助
OUT D0.05  ; 整机复位启动
; rung 4
LD D0.05  ; 整机复位启动
OR D1.00  ; 整机复位开始
ANDNOT D0.04  ; 报警清除&错误复位
ANDNOT D0.04  ; 报警清除&错误复位
ANDNOT D0.10  ; 机台有故障
ANDNOT T0005  ; 整机在初始位延时
OUT D1.00  ; 整机复位开始
; rung 5
LD D0.05  ; 整机复位启动
OR D1.01  ; 整机复位开始延时
ANDNOT D0.04  ; 报警清除&错误复位
ANDNOT D0.04  ; 报警清除&错误复位
ANDNOT T0023  ; 整机在初始位延时
OUT D1.01  ; 整机复位开始延时
; rung 6
LD D1.00  ; 整机复位开始
OUT W40.10  ; 进料机构复位
OUT W50.10  ; 上下料机构手复位
OUT W60.00  ; 腔体机构手复位
OUT W70.00  ; 出料机构手复位

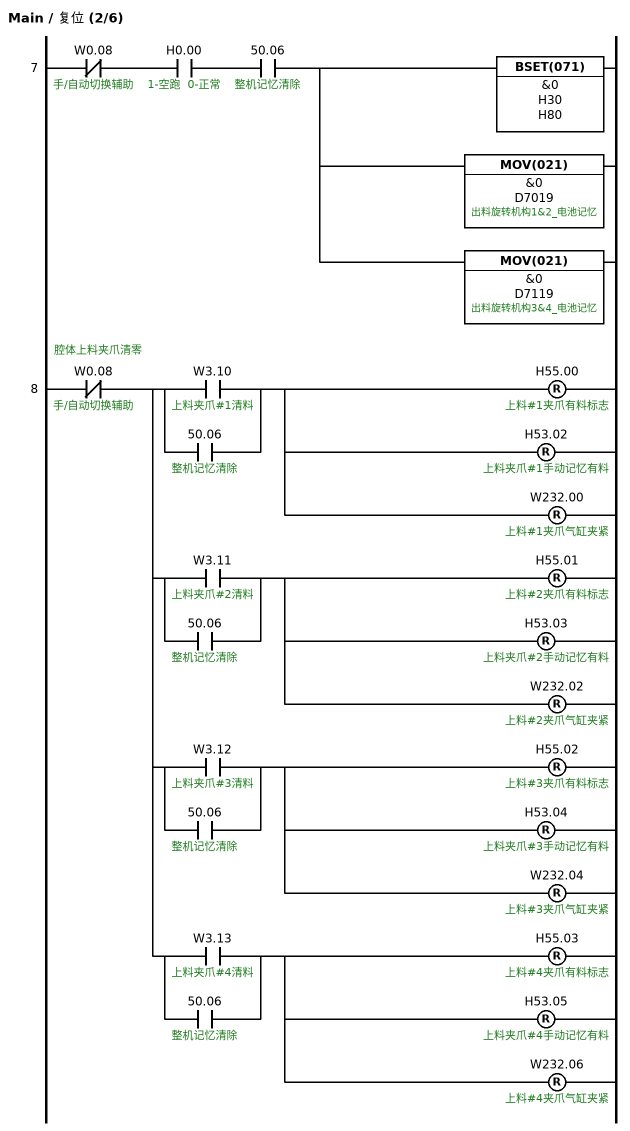
; rung 7
LDNOT W0.08  ; 手/自动切换辅助
AND H0.00  ; 1-空跑  0-正常
AND 50.06  ; 整机记忆清除
BSET(071) &0 H30 H80
MOV(021) &0 D7019  ; 出料旋转机构1&2_电池记忆
MOV(021) &0 D7119  ; 出料旋转机构3&4_电池记忆
; rung 8: 腔体上料夹爪清零
LDNOT W0.08  ; 手/自动切换辅助
OUT TR0
LD W3.10  ; 上料夹爪#1清料
OR 50.06  ; 整机记忆清除
ANDLD
RSET H55.00  ; 上料#1夹爪有料标志
RSET H53.02  ; 上料夹爪#1手动记忆有料
RSET W232.00  ; 上料#1夹爪气缸夹紧
LD TR0
LD W3.11  ; 上料夹爪#2清料
OR 50.06  ; 整机记忆清除
ANDLD
RSET H55.01  ; 上料#2夹爪有料标志
RSET H53.03  ; 上料夹爪#2手动记忆有料
RSET W232.02  ; 上料#2夹爪气缸夹紧
LD TR0
LD W3.12  ; 上料夹爪#3清料
OR 50.06  ; 整机记忆清除
ANDLD
RSET H55.02  ; 上料#3夹爪有料标志
RSET H53.04  ; 上料夹爪#3手动记忆有料
RSET W232.04  ; 上料#3夹爪气缸夹紧
LD TR0
LD W3.13  ; 上料夹爪#4清料
OR 50.06  ; 整机记忆清除
ANDLD
RSET H55.03  ; 上料#4夹爪有料标志
RSET H53.05  ; 上料夹爪#4手动记忆有料
RSET W232.06  ; 上料#4夹爪气缸夹紧

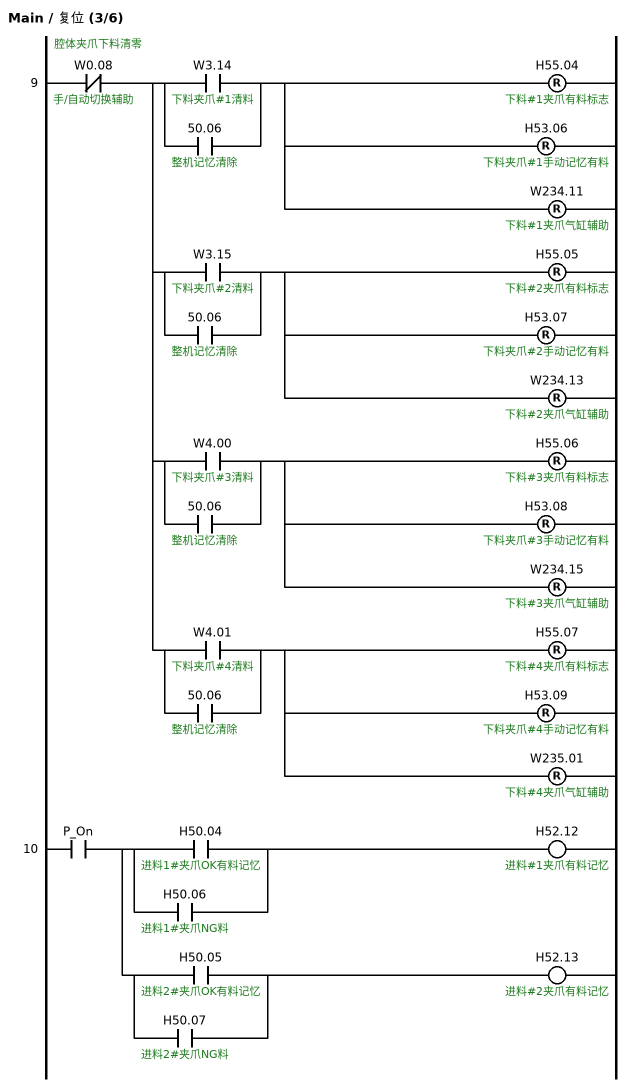
; rung 9: 腔体夹爪下料清零
LDNOT W0.08  ; 手/自动切换辅助
OUT TR0
LD W3.14  ; 下料夹爪#1清料
OR 50.06  ; 整机记忆清除
ANDLD
RSET H55.04  ; 下料#1夹爪有料标志
RSET H53.06  ; 下料夹爪#1手动记忆有料
RSET W234.11  ; 下料#1夹爪气缸辅助
LD TR0
LD W3.15  ; 下料夹爪#2清料
OR 50.06  ; 整机记忆清除
ANDLD
RSET H55.05  ; 下料#2夹爪有料标志
RSET H53.07  ; 下料夹爪#2手动记忆有料
RSET W234.13  ; 下料#2夹爪气缸辅助
LD TR0
LD W4.00  ; 下料夹爪#3清料
OR 50.06  ; 整机记忆清除
ANDLD
RSET H55.06  ; 下料#3夹爪有料标志
RSET H53.08  ; 下料夹爪#3手动记忆有料
RSET W234.15  ; 下料#3夹爪气缸辅助
LD TR0
LD W4.01  ; 下料夹爪#4清料
OR 50.06  ; 整机记忆清除
ANDLD
RSET H55.07  ; 下料#4夹爪有料标志
RSET H53.09  ; 下料夹爪#4手动记忆有料
RSET W235.01  ; 下料#4夹爪气缸辅助
; rung 10
LD P_On
OUT TR0
LD H50.04  ; 进料1#夹爪OK有料记忆
OR H50.06  ; 进料1#夹爪NG料
ANDLD
OUT H52.12  ; 进料#1夹爪有料记忆
LD TR0
LD H50.05  ; 进料2#夹爪OK有料记忆
OR H50.07  ; 进料2#夹爪NG料
ANDLD
OUT H52.13  ; 进料#2夹爪有料记忆

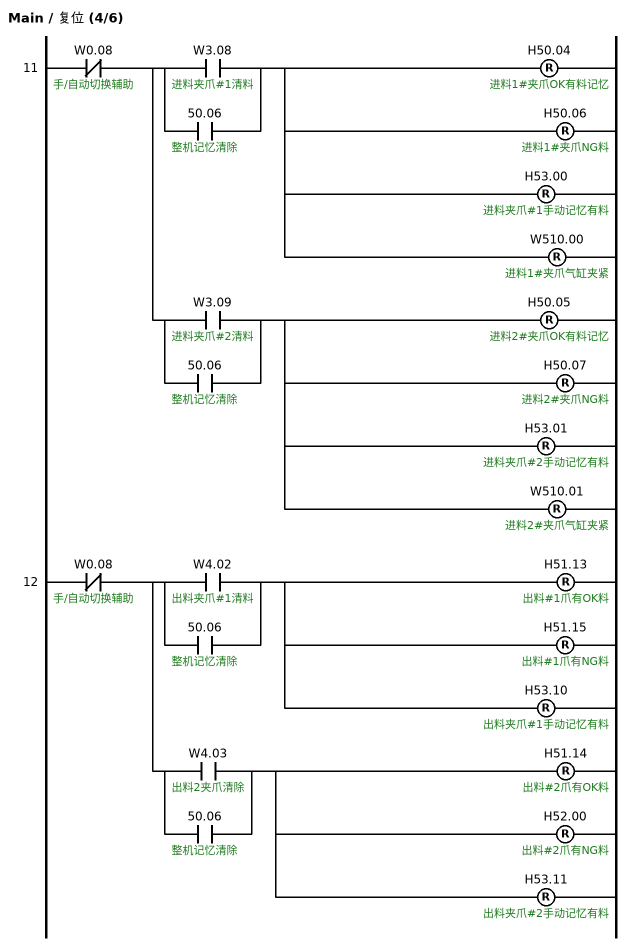
; rung 11
LDNOT W0.08  ; 手/自动切换辅助
OUT TR0
LD W3.08  ; 进料夹爪#1清料
OR 50.06  ; 整机记忆清除
ANDLD
RSET H50.04  ; 进料1#夹爪OK有料记忆
RSET H50.06  ; 进料1#夹爪NG料
RSET H53.00  ; 进料夹爪#1手动记忆有料
RSET W510.00  ; 进料1#夹爪气缸夹紧
LD TR0
LD W3.09  ; 进料夹爪#2清料
OR 50.06  ; 整机记忆清除
ANDLD
RSET H50.05  ; 进料2#夹爪OK有料记忆
RSET H50.07  ; 进料2#夹爪NG料
RSET H53.01  ; 进料夹爪#2手动记忆有料
RSET W510.01  ; 进料2#夹爪气缸夹紧
; rung 12
LDNOT W0.08  ; 手/自动切换辅助
OUT TR0
LD W4.02  ; 出料夹爪#1清料
OR 50.06  ; 整机记忆清除
ANDLD
RSET H51.13  ; 出料#1爪有OK料
RSET H51.15  ; 出料#1爪有NG料
RSET H53.10  ; 出料夹爪#1手动记忆有料
LD TR0
LD W4.03  ; 出料2夹爪清除
OR 50.06  ; 整机记忆清除
ANDLD
RSET H51.14  ; 出料#2爪有OK料
RSET H52.00  ; 出料#2爪有NG料
RSET H53.11  ; 出料夹爪#2手动记忆有料

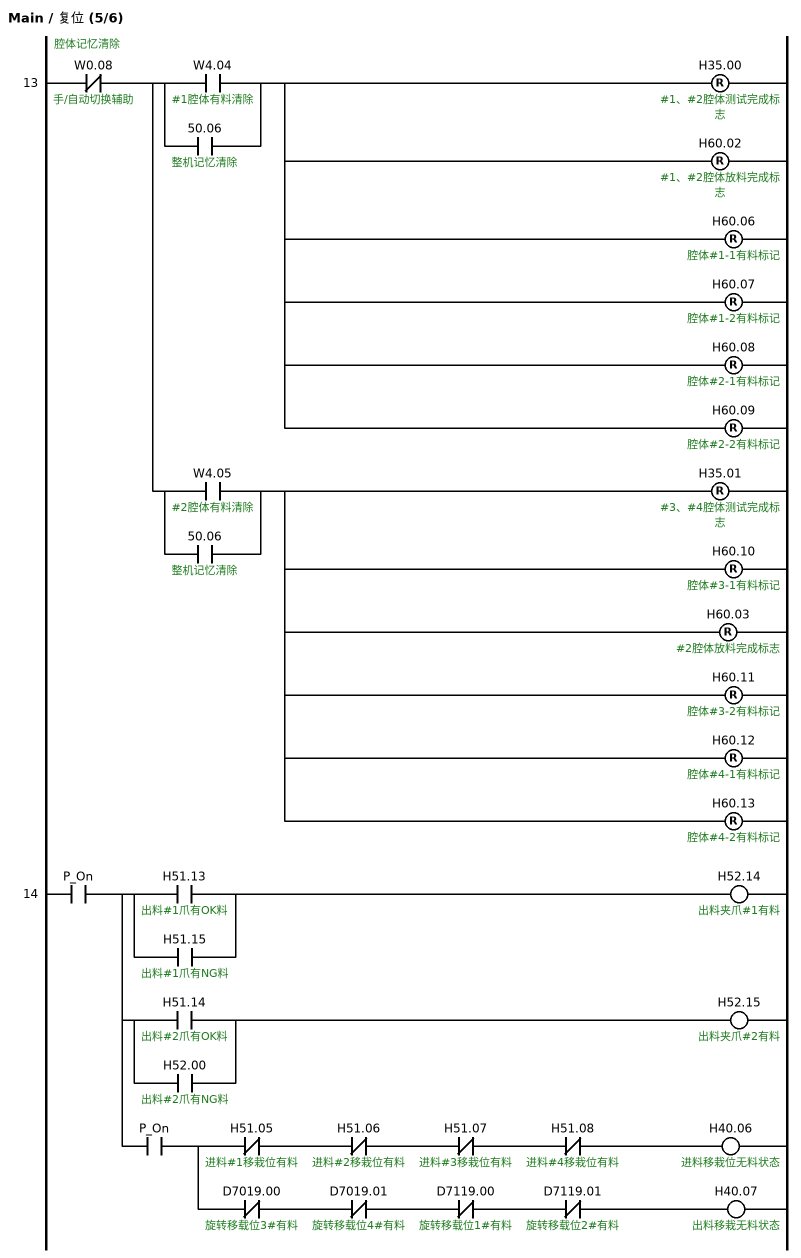
; rung 13: 腔体记忆清除
LDNOT W0.08  ; 手/自动切换辅助
OUT TR0
LD W4.04  ; #1腔体有料清除
OR 50.06  ; 整机记忆清除
ANDLD
RSET H35.00  ; #1、#2腔体测试完成标志
RSET H60.02  ; #1、#2腔体放料完成标志
RSET H60.06  ; 腔体#1-1有料标记
RSET H60.07  ; 腔体#1-2有料标记
RSET H60.08  ; 腔体#2-1有料标记
RSET H60.09  ; 腔体#2-2有料标记
LD TR0
LD W4.05  ; #2腔体有料清除
OR 50.06  ; 整机记忆清除
ANDLD
RSET H35.01  ; #3、#4腔体测试完成标志
RSET H60.10  ; 腔体#3-1有料标记
RSET H60.03  ; #2腔体放料完成标志
RSET H60.11  ; 腔体#3-2有料标记
RSET H60.12  ; 腔体#4-1有料标记
RSET H60.13  ; 腔体#4-2有料标记
; rung 14
LD P_On
OUT TR0
LD H51.13  ; 出料#1爪有OK料
OR H51.15  ; 出料#1爪有NG料
ANDLD
OUT H52.14  ; 出料夹爪#1有料
LD TR0
LD H51.14  ; 出料#2爪有OK料
OR H52.00  ; 出料#2爪有NG料
ANDLD
OUT H52.15  ; 出料夹爪#2有料
LD TR0
AND P_On
OUT TR0
ANDNOT H51.05  ; 进料#1移栽位有料
ANDNOT H51.06  ; 进料#2移栽位有料
ANDNOT H51.07  ; 进料#3移栽位有料
ANDNOT H51.08  ; 进料#4移栽位有料
OUT H40.06  ; 进料移栽位无料状态
LD TR0
ANDNOT D7019.00  ; 旋转移载位3#有料
ANDNOT D7019.01  ; 旋转移载位4#有料
ANDNOT D7119.00  ; 旋转移载位1#有料
ANDNOT D7119.01  ; 旋转移载位2#有料
OUT H40.07  ; 出料移栽无料状态

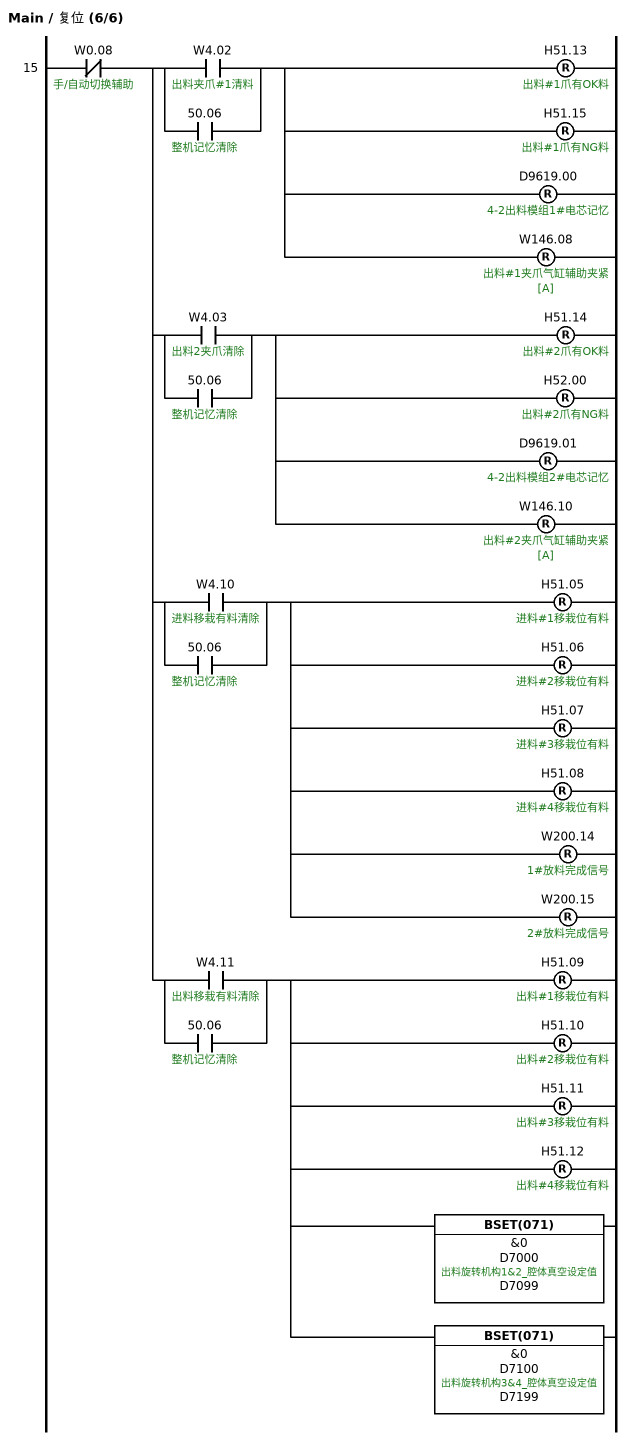
; rung 15
LDNOT W0.08  ; 手/自动切换辅助
OUT TR0
LD W4.02  ; 出料夹爪#1清料
OR 50.06  ; 整机记忆清除
ANDLD
RSET H51.13  ; 出料#1爪有OK料
RSET H51.15  ; 出料#1爪有NG料
RSET D9619.00  ; 4-2出料模组1#电芯记忆
RSET W146.08  ; 出料#1夹爪气缸辅助夹紧[A]
LD TR0
LD W4.03  ; 出料2夹爪清除
OR 50.06  ; 整机记忆清除
ANDLD
RSET H51.14  ; 出料#2爪有OK料
RSET H52.00  ; 出料#2爪有NG料
RSET D9619.01  ; 4-2出料模组2#电芯记忆
RSET W146.10  ; 出料#2夹爪气缸辅助夹紧[A]
LD TR0
LD W4.10  ; 进料移栽有料清除
OR 50.06  ; 整机记忆清除
ANDLD
RSET H51.05  ; 进料#1移栽位有料
RSET H51.06  ; 进料#2移栽位有料
RSET H51.07  ; 进料#3移栽位有料
RSET H51.08  ; 进料#4移栽位有料
RSET W200.14  ; 1#放料完成信号
RSET W200.15  ; 2#放料完成信号
LD TR0
LD W4.11  ; 出料移栽有料清除
OR 50.06  ; 整机记忆清除
ANDLD
RSET H51.09  ; 出料#1移栽位有料
RSET H51.10  ; 出料#2移栽位有料
RSET H51.11  ; 出料#3移栽位有料
RSET H51.12  ; 出料#4移栽位有料
BSET(071) &0 D7000 D7099  ; 出料旋转机构1&2_腔体真空设定值
BSET(071) &0 D7100 D7199  ; 出料旋转机构3&4_腔体真空设定值

### Section 指示灯输出

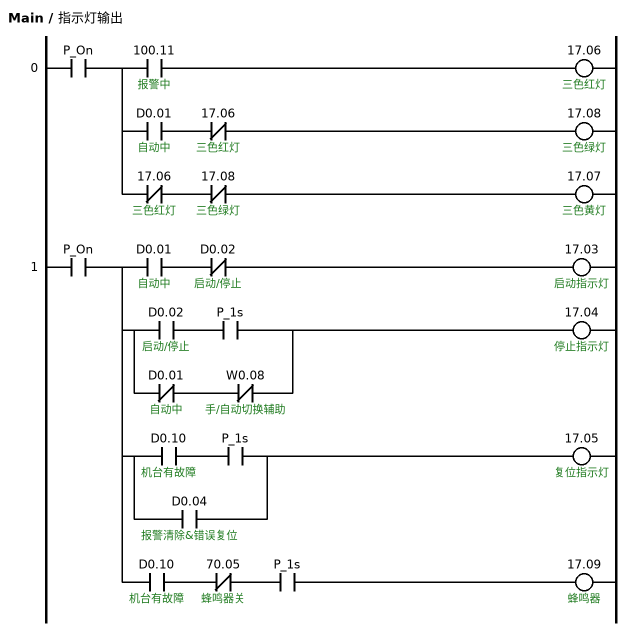
; rung 0
LD P_On
OUT TR0
AND 100.11  ; 报警中
OUT 17.06  ; 三色红灯
LD TR0
AND D0.01  ; 自动中
ANDNOT 17.06  ; 三色红灯
OUT 17.08  ; 三色绿灯
LD TR0
ANDNOT 17.06  ; 三色红灯
ANDNOT 17.08  ; 三色绿灯
OUT 17.07  ; 三色黄灯
; rung 1
LD P_On
OUT TR0
AND D0.01  ; 自动中
ANDNOT D0.02  ; 启动/停止
OUT 17.03  ; 启动指示灯
LD TR0
LD D0.02  ; 启动/停止
AND P_1s
LDNOT D0.01  ; 自动中
ANDNOT W0.08  ; 手/自动切换辅助
ORLD
ANDLD
OUT 17.04  ; 停止指示灯
LD TR0
LD D0.10  ; 机台有故障
AND P_1s
OR D0.04  ; 报警清除&错误复位
ANDLD
OUT 17.05  ; 复位指示灯
LD TR0
AND D0.10  ; 机台有故障
ANDNOT 70.05  ; 蜂鸣器关
AND P_1s
OUT 17.09  ; 蜂鸣器

### Section PC交互

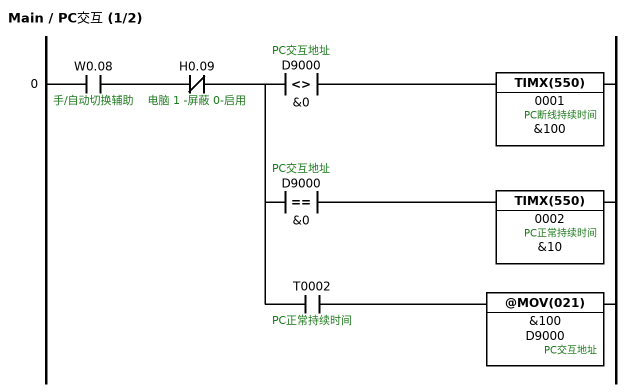
; rung 0
LD W0.08  ; 手/自动切换辅助
ANDNOT H0.09  ; 电脑 1 -屏蔽 0-启用
OUT TR0
AND<>(305) D9000 &0  ; PC交互地址
TIMX(550) 0001 &100  ; PC断线持续时间
LD TR0
AND=(300) D9000 &0  ; PC交互地址
TIMX(550) 0002 &10  ; PC正常持续时间
LD TR0
AND T0002  ; PC正常持续时间
@MOV(021) &100 D9000  ; PC交互地址

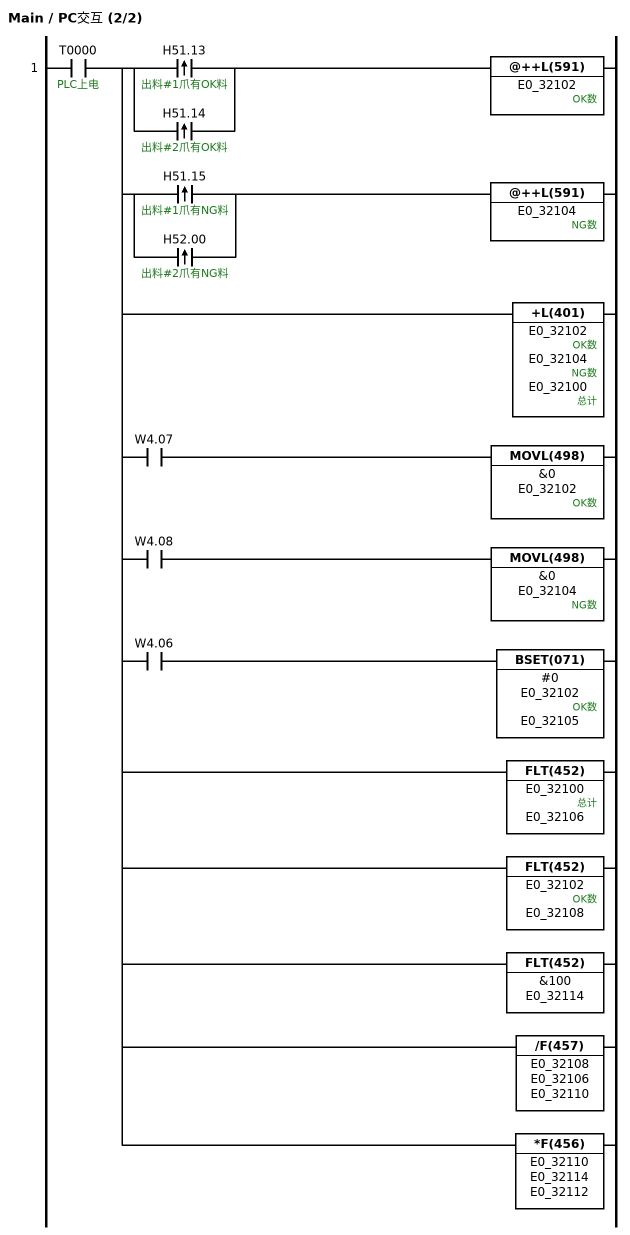
; rung 1
LD T0000  ; PLC上电
OUT TR0
@LD H51.13  ; 出料#1爪有OK料
@OR H51.14  ; 出料#2爪有OK料
ANDLD
@++L(591) E0_32102  ; OK数
LD TR0
@LD H51.15  ; 出料#1爪有NG料
@OR H52.00  ; 出料#2爪有NG料
ANDLD
@++L(591) E0_32104  ; NG数
LD TR0
+L(401) E0_32102 E0_32104 E0_32100  ; OK数, NG数, 总计
AND W4.07
MOVL(498) &0 E0_32102  ; OK数
LD TR0
AND W4.08
MOVL(498) &0 E0_32104  ; NG数
LD TR0
AND W4.06
BSET(071) #0 E0_32102 E0_32105  ; OK数
LD TR0
FLT(452) E0_32100 E0_32106  ; 总计
FLT(452) E0_32102 E0_32108  ; OK数
FLT(452) &100 E0_32114
/F(457) E0_32108 E0_32106 E0_32110
*F(456) E0_32110 E0_32114 E0_32112

### Section END
; rung 0
END(001)

## Program 进料机构 (cyclic task 1)

### Section 安全限制条件

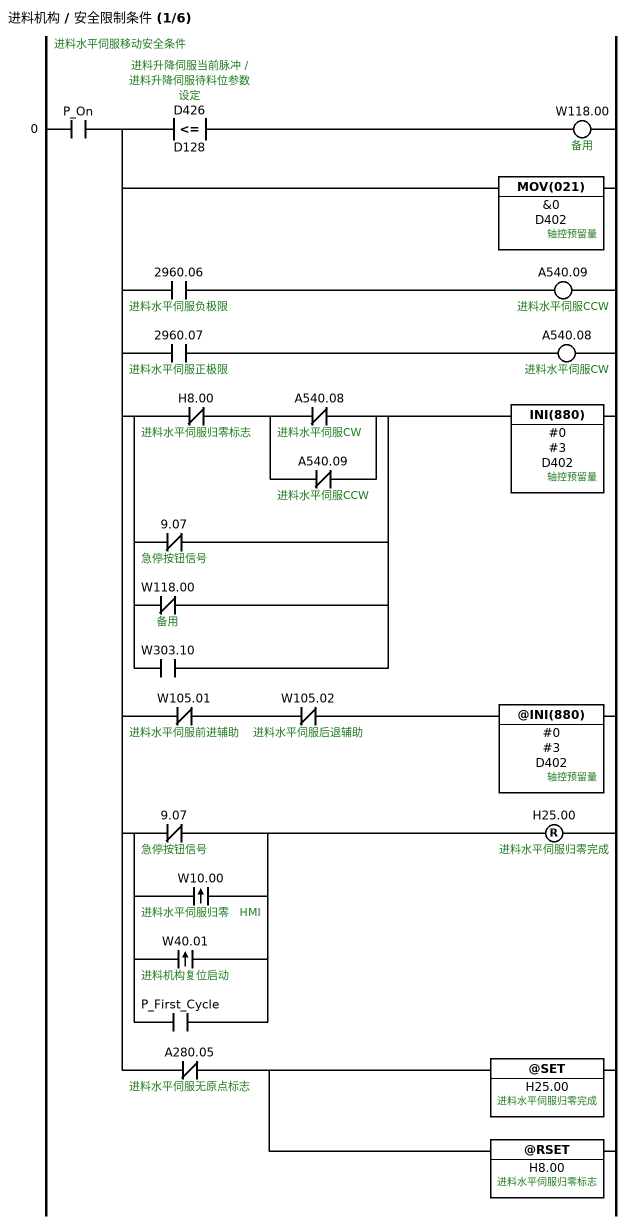
; rung 0: 进料水平伺服移动安全条件
LD P_On
OUT TR0
AND<=SL(318) D426 D128  ; 进料升降伺服当前脉冲, 进料升降伺服待料位参数设定
OUT W118.00  ; 备用
LD TR0
MOV(021) &0 D402  ; 轴控预留量
AND 2960.06  ; 进料水平伺服负极限
OUT A540.09  ; 进料水平伺服CCW
LD TR0
AND 2960.07  ; 进料水平伺服正极限
OUT A540.08  ; 进料水平伺服CW
LD TR0
LDNOT H8.00  ; 进料水平伺服归零标志
LDNOT A540.08  ; 进料水平伺服CW
ORNOT A540.09  ; 进料水平伺服CCW
ANDLD
ORNOT 9.07  ; 急停按钮信号
ORNOT W118.00  ; 备用
OR W303.10
ANDLD
INI(880) #0 #3 D402  ; 轴控预留量
LD TR0
ANDNOT W105.01  ; 进料水平伺服前进辅助
ANDNOT W105.02  ; 进料水平伺服后退辅助
@INI(880) #0 #3 D402  ; 轴控预留量
LD TR0
LDNOT 9.07  ; 急停按钮信号
@OR W10.00  ; 进料水平伺服归零   HMI
@OR W40.01  ; 进料机构复位启动
OR P_First_Cycle
ANDLD
RSET H25.00  ; 进料水平伺服归零完成
LD TR0
ANDNOT A280.05  ; 进料水平伺服无原点标志
@SET H25.00  ; 进料水平伺服归零完成
@RSET H8.00  ; 进料水平伺服归零标志

